SUBAPPLICATION Uebung_080f_AX (* Beispiel für E_CTU *)
  (* Standard: 61499-2; Description: Copyright (c) 2023 Meisterschulen am Ostbahnhof This program and the accompanying materials are made available under the terms of the Eclipse Public License 2.0 which is available at https://www.eclipse.org/legal/epl-2.0/ SPDX-License-Identifier: EPL-2.0 *)
  (* Version 1.0, 2023-10-23, Franz Höpfinger, Meisterschulen am Ostbahnhof, initial API and implementation and/or initial documentation *)
  PACKAGE Uebungen;
  IMPORT Uebungen::const::UT::Horse::DefaultPool_Horse::ObjectPointer_Horse;
  IMPORT Uebungen::const::UT::Horse::DefaultPool_Horse::frame_00;
  IMPORT Uebungen::const::UT::Horse::DefaultPool_Horse::frame_01;
  IMPORT Uebungen::const::UT::Horse::DefaultPool_Horse::frame_02;
  IMPORT Uebungen::const::UT::Horse::DefaultPool_Horse::frame_03;
  IMPORT Uebungen::const::UT::Horse::DefaultPool_Horse::frame_04;
  IMPORT Uebungen::const::UT::Horse::DefaultPool_Horse::frame_05;
  IMPORT Uebungen::const::UT::Horse::DefaultPool_Horse::frame_06;
  IMPORT Uebungen::const::UT::Horse::DefaultPool_Horse::frame_07;
  IMPORT Uebungen::const::UT::Horse::DefaultPool_Horse::frame_08;
  IMPORT Uebungen::const::UT::Horse::DefaultPool_Horse::frame_09;
  IMPORT Uebungen::const::UT::Horse::DefaultPool_Horse::frame_10;
  IMPORT Uebungen::const::UT::Horse::DefaultPool_Horse::frame_11;
  IMPORT Uebungen::const::UT::Horse::DefaultPool_Horse::frame_12;
  IMPORT Uebungen::const::UT::Horse::DefaultPool_Horse::frame_13;
  IMPORT Uebungen::const::UT::Horse::DefaultPool_Horse::frame_14;
  IMPORT Uebungen::const::UT::Horse::DefaultPool_Horse::frame_15;
  IMPORT Uebungen::const::UT::Horse::DefaultPool_Horse::frame_16;
  IMPORT Uebungen::const::UT::Horse::DefaultPool_Horse::frame_17;
  IMPORT Uebungen::const::UT::Horse::DefaultPool_Horse::frame_18;
  IMPORT Uebungen::const::UT::Horse::DefaultPool_Horse::frame_19;
  IMPORT Uebungen::const::UT::Horse::DefaultPool_Horse::frame_20;
  IMPORT Uebungen::const::UT::Horse::DefaultPool_Horse::frame_21;
  IMPORT Uebungen::const::UT::Horse::DefaultPool_Horse::frame_22;
  IMPORT Uebungen::const::UT::Horse::DefaultPool_Horse::frame_23;
  IMPORT Uebungen::const::UT::Horse::DefaultPool_Horse::frame_24;
  IMPORT Uebungen::const::UT::Horse::DefaultPool_Horse::frame_25;
  IMPORT Uebungen::const::UT::Horse::DefaultPool_Horse::frame_26;
  IMPORT Uebungen::const::UT::Horse::DefaultPool_Horse::frame_27;
  IMPORT Uebungen::const::UT::Horse::DefaultPool_Horse::frame_28;
  IMPORT Uebungen::const::UT::Horse::DefaultPool_Horse::frame_29;
  IMPORT Uebungen::const::UT::Horse::DefaultPool_Horse::frame_30;
  IMPORT Uebungen::const::UT::Horse::DefaultPool_Horse::frame_31;
  IMPORT logiBUS::io::DI::logiBUS_DI::Input_I1;
  IMPORT logiBUS::io::DI::logiBUS_DI::Input_I2;
  IMPORT logiBUS::io::DI::logiBUS_DI_Events::BUTTON_SINGLE_CLICK;
  IMPORT logiBUS::io::DQ::logiBUS_DO::Output_Q1;
  FBS
    DigitalOutput_Q1 : logiBUS::io::DQ::logiBUS_QXA(QI := TRUE, Output := Output_Q1);
    DigitalInput_CLK_I1 : logiBUS::io::DI::logiBUS_IE(QI := TRUE, Input := Input_I1, InputEvent := BUTTON_SINGLE_CLICK);
    AUI_CTU : adapter::events::unidirectional::AUI_CTU;
    DigitalInput_CLK_I2 : logiBUS::io::DI::logiBUS_IE(QI := TRUE, Input := Input_I2, InputEvent := BUTTON_SINGLE_CLICK);
    initval_00 : adapter::types::unidirectional::AUDI::initval::initval_AUDI(INIT_VAL := frame_00);
    initval_01 : adapter::types::unidirectional::AUDI::initval::initval_AUDI(INIT_VAL := frame_01);
    initval_02 : adapter::types::unidirectional::AUDI::initval::initval_AUDI(INIT_VAL := frame_02);
    initval_03 : adapter::types::unidirectional::AUDI::initval::initval_AUDI(INIT_VAL := frame_03);
    initval_04 : adapter::types::unidirectional::AUDI::initval::initval_AUDI(INIT_VAL := frame_04);
    initval_05 : adapter::types::unidirectional::AUDI::initval::initval_AUDI(INIT_VAL := frame_05);
    initval_06 : adapter::types::unidirectional::AUDI::initval::initval_AUDI(INIT_VAL := frame_06);
    initval_07 : adapter::types::unidirectional::AUDI::initval::initval_AUDI(INIT_VAL := frame_07);
    initval_08 : adapter::types::unidirectional::AUDI::initval::initval_AUDI(INIT_VAL := frame_08);
    initval_09 : adapter::types::unidirectional::AUDI::initval::initval_AUDI(INIT_VAL := frame_09);
    initval_10 : adapter::types::unidirectional::AUDI::initval::initval_AUDI(INIT_VAL := frame_10);
    initval_11 : adapter::types::unidirectional::AUDI::initval::initval_AUDI(INIT_VAL := frame_11);
    initval_12 : adapter::types::unidirectional::AUDI::initval::initval_AUDI(INIT_VAL := frame_12);
    initval_13 : adapter::types::unidirectional::AUDI::initval::initval_AUDI(INIT_VAL := frame_13);
    initval_14 : adapter::types::unidirectional::AUDI::initval::initval_AUDI(INIT_VAL := frame_14);
    initval_15 : adapter::types::unidirectional::AUDI::initval::initval_AUDI(INIT_VAL := frame_15);
    initval_16 : adapter::types::unidirectional::AUDI::initval::initval_AUDI(INIT_VAL := frame_16);
    initval_17 : adapter::types::unidirectional::AUDI::initval::initval_AUDI(INIT_VAL := frame_17);
    initval_18 : adapter::types::unidirectional::AUDI::initval::initval_AUDI(INIT_VAL := frame_18);
    initval_19 : adapter::types::unidirectional::AUDI::initval::initval_AUDI(INIT_VAL := frame_19);
    initval_20 : adapter::types::unidirectional::AUDI::initval::initval_AUDI(INIT_VAL := frame_20);
    initval_21 : adapter::types::unidirectional::AUDI::initval::initval_AUDI(INIT_VAL := frame_21);
    initval_22 : adapter::types::unidirectional::AUDI::initval::initval_AUDI(INIT_VAL := frame_22);
    initval_23 : adapter::types::unidirectional::AUDI::initval::initval_AUDI(INIT_VAL := frame_23);
    initval_24 : adapter::types::unidirectional::AUDI::initval::initval_AUDI(INIT_VAL := frame_24);
    initval_25 : adapter::types::unidirectional::AUDI::initval::initval_AUDI(INIT_VAL := frame_25);
    initval_26 : adapter::types::unidirectional::AUDI::initval::initval_AUDI(INIT_VAL := frame_26);
    initval_27 : adapter::types::unidirectional::AUDI::initval::initval_AUDI(INIT_VAL := frame_27);
    initval_28 : adapter::types::unidirectional::AUDI::initval::initval_AUDI(INIT_VAL := frame_28);
    initval_29 : adapter::types::unidirectional::AUDI::initval::initval_AUDI(INIT_VAL := frame_29);
    initval_30 : adapter::types::unidirectional::AUDI::initval::initval_AUDI(INIT_VAL := frame_30);
    initval_31 : adapter::types::unidirectional::AUDI::initval::initval_AUDI(INIT_VAL := frame_31);
    AUDI_AUI_MUX_32 : adapter::selection::unidirectional::AUDI_AUI_MUX_32;
    Q_NumericValue_1 : isobus::UT::Q::Q_NumericValue_AUDI(u16ObjId := ObjectPointer_Horse);
  END_FBS
  EVENT_CONNECTIONS
    DigitalInput_CLK_I1.IND TO AUI_CTU.CU;
    DigitalInput_CLK_I2.IND TO AUI_CTU.R;
  END_CONNECTIONS
  ADAPTER_CONNECTIONS
    AUI_CTU.Q TO DigitalOutput_Q1.OUT;
    AUI_CTU.CV TO AUDI_AUI_MUX_32.K;
    initval_00.OUT TO AUDI_AUI_MUX_32.IN1;
    initval_01.OUT TO AUDI_AUI_MUX_32.IN2;
    initval_02.OUT TO AUDI_AUI_MUX_32.IN3;
    initval_03.OUT TO AUDI_AUI_MUX_32.IN4;
    initval_04.OUT TO AUDI_AUI_MUX_32.IN5;
    initval_05.OUT TO AUDI_AUI_MUX_32.IN6;
    initval_06.OUT TO AUDI_AUI_MUX_32.IN7;
    initval_07.OUT TO AUDI_AUI_MUX_32.IN8;
    initval_08.OUT TO AUDI_AUI_MUX_32.IN9;
    initval_09.OUT TO AUDI_AUI_MUX_32.IN10;
    initval_10.OUT TO AUDI_AUI_MUX_32.IN11;
    initval_11.OUT TO AUDI_AUI_MUX_32.IN12;
    initval_12.OUT TO AUDI_AUI_MUX_32.IN13;
    initval_13.OUT TO AUDI_AUI_MUX_32.IN14;
    initval_14.OUT TO AUDI_AUI_MUX_32.IN15;
    initval_15.OUT TO AUDI_AUI_MUX_32.IN16;
    initval_16.OUT TO AUDI_AUI_MUX_32.IN17;
    initval_17.OUT TO AUDI_AUI_MUX_32.IN18;
    initval_18.OUT TO AUDI_AUI_MUX_32.IN19;
    initval_19.OUT TO AUDI_AUI_MUX_32.IN20;
    initval_20.OUT TO AUDI_AUI_MUX_32.IN21;
    initval_21.OUT TO AUDI_AUI_MUX_32.IN22;
    initval_22.OUT TO AUDI_AUI_MUX_32.IN23;
    initval_23.OUT TO AUDI_AUI_MUX_32.IN24;
    initval_24.OUT TO AUDI_AUI_MUX_32.IN25;
    initval_25.OUT TO AUDI_AUI_MUX_32.IN26;
    initval_26.OUT TO AUDI_AUI_MUX_32.IN27;
    initval_27.OUT TO AUDI_AUI_MUX_32.IN28;
    initval_28.OUT TO AUDI_AUI_MUX_32.IN29;
    initval_29.OUT TO AUDI_AUI_MUX_32.IN30;
    initval_30.OUT TO AUDI_AUI_MUX_32.IN31;
    initval_31.OUT TO AUDI_AUI_MUX_32.IN32;
    AUDI_AUI_MUX_32.OUT TO Q_NumericValue_1.u32NewValue;
  END_CONNECTIONS
END_SUBAPPLICATION
